// TIA Portal project "2022.06.14_通信方式" (V17)

(* hardware
DEVICE "S7-1200 station_1"  S7-1200 Station
   slot 0: "Rack_0"  S7-1200 Rack  Rack  V1.0
   slot 1: "PLC_1"  CPU 1212C DC/DC/DC  6ES7 212-1AE40-0XB0  V4.5
   slot 2: "AI 4x13BIT/AQ 2x14BIT_1"  SM 1234 AI4/AQ2  6ES7 234-4HE30-0XB0  V1.0
*)

// ===== PLC "PLC_1"  CPU 1212C DC/DC/DC =====

VAR_GLOBAL   // PLC tag table "默认变量表"
   "液位测量" AT %IW96 : Word;
   "百分比" AT %MD40 : DWord;
   "模拟量输出通道" AT %MD44 : UDInt;
   "所需频率(1)" AT %MD0 : Real;
   "压力2模拟输入通道" AT %IW100 : Int;
   "液位" AT %MD4 : Real;
   "频率" AT %MD8 : Real;
   "Tag_2" AT %MD12 : Real;
   "模拟量输出" AT %QW96 : Int;
   "设定液位值" AT %MD20 : Real;
   "实际液位值" AT %MD24 : Real;
   "轴_1_脉冲" AT %Q0.0 : Bool;
   "轴_1_方向" AT %Q0.1 : Bool;
   "轴_1_LowHwLimitSwitch" AT %I0.0 : Bool;
   "轴_1_HighHwLimitSwitch" AT %I0.1 : Bool;
   "轴_1_PassiveHomingSwitch" AT %I0.2 : Bool;
   "轴_1_归位开关" AT %I0.3 : Bool;
   "启用轴" AT %M0.0 : Bool;
   "完成位" AT %M0.1 : Bool;
   "Tag_1" AT %M0.2 : Bool;
   "回原点" AT %I1.0 : Bool;
   "Tag_3" AT %M0.4 : Bool;
   "Tag_4" AT %M0.5 : Bool;
   "Tag_5" AT %M0.3 : Bool;
   "触发绝对定位" AT %I1.1 : Bool;
   "Tag_7" AT %M0.6 : Bool;
   "指定位置" AT %MD30 : Real;
   "指定速度" AT %MD34 : Real;
   "Tag_6" AT %M0.7 : Bool;
   "Tag_8" AT %I1.2 : Bool;
   "Tag_9" AT %M1.0 : Bool;
   "触发相对位移指令" AT %I1.3 : Bool;
   "Tag_11" AT %M1.1 : Bool;
   "相对位置" AT %MD28 : Real;
   "速度" AT %MD32 : Real;
   "触发恒速" AT %I0.4 : Bool;
   "Tag_10" AT %M1.2 : Bool;
   "Tag_12" AT %MD36 : Real;
   "Tag_13" AT %I1.5 : Bool;
   "Tag_14" AT %M1.3 : Bool;
   "正点动" AT %I1.6 : Bool;
   "反点动" AT %I1.7 : Bool;
   "System_Byte" AT %MB100 : Byte;
   "FirstScan" AT %M100.0 : Bool;
   "DiagStatusUpdate" AT %M100.1 : Bool;
   "AlwaysTRUE" AT %M100.2 : Bool;
   "AlwaysFALSE" AT %M100.3 : Bool;
   "Tag_15" AT %M10.0 : Bool;
   "Tag_16" AT %M70.0 : Bool;
   "Tag_17" AT %M70.1 : Bool;
   "Tag_18" AT %M70.2 : Bool;
   "Clock_Byte" AT %MB10 : Byte;
   "Clock_10Hz" AT %M10.0 : Bool;
   "Clock_5Hz" AT %M10.1 : Bool;
   "Clock_2.5Hz" AT %M10.2 : Bool;
   "Clock_2Hz" AT %M10.3 : Bool;
   "Clock_1.25Hz" AT %M10.4 : Bool;
   "Clock_1Hz" AT %M10.5 : Bool;
   "Clock_0.625Hz" AT %M10.6 : Bool;
   "Clock_0.5Hz" AT %M10.7 : Bool;
END_VAR

DATA_BLOCK "发送数据"   // DB15
{ S7_Optimized_Access := 'FALSE' }
VERSION : 0.1
   VAR
      发送1 : Real;
      发送2 : Real;
      发送3 : Real;
      发送4 : Real;
   END_VAR
BEGIN
END_DATA_BLOCK

DATA_BLOCK "接收"   // DB18
{ S7_Optimized_Access := 'FALSE' }
VERSION : 0.1
   VAR
      接受1 : Real;
      接受2 : Real;
      接受3 : Real;
      接受4 : Real;
   END_VAR
BEGIN
END_DATA_BLOCK

// folder: System blocks/Program resources

DATA_BLOCK "IEC_Timer_0_DB"   // DB13
{ S7_Optimized_Access := 'TRUE' }
AUTHOR : Simatic
FAMILY : IEC
NAME : IEC_TMR
VERSION : 1.0
// stored: InstanceOfName IEC_TIMER
"IEC_TIMER"
BEGIN
END_DATA_BLOCK

// folder: (top level)

DATA_BLOCK "轴_1"   // DB2, Motion_DB
{ S7_Optimized_Access := 'TRUE' }
AUTHOR : SIMATIC
FAMILY : BasicMC
NAME : TO_PosAx
VERSION : 8.0
// stored: InstanceOfName TO_PositioningAxis
"TO_PositioningAxis"
BEGIN
   // Axis.HomingReferencePointSwitch_AddressCU = %I0.3
   // Axis.LengthUnitNormalized.Distance = 1013
   // Axis.PositionLimitsMax_AddressCU = %I0.1
   // Axis.PositionLimitsMin_AddressCU = %I0.0
   // Axis.OnlinePtoModeCU = 16#0000_0002
   // Axis.DirectionOutputEnabledCU = TRUE
   // Axis.SelectedChannel2EnumCU = %Q0.1
   // Axis.SelectedChannel1EnumCU = %Q0.0
   // Pulse.MinDeltaDeltaFrequencyCU = 0.004
   // Pulse.MaxDeltaDeltaFrequencyCU = 1.0E+10
   // Pulse.MinDeltaFrequencyCU = 0.005
   // Pulse.MaxDeltaFrequencyCU = 9.5E+9
   // Pulse.MinFrequencyCU = 1.0
   // Pulse.MaxFrequencyCU = 100000.0
   // Pulse.OutputSourceCU = 16#0000_0000
   // Axis.SelectPTO = 0
END_DATA_BLOCK

ORGANIZATION_BLOCK "Main"   // OB1, LAD, ProgramCycle
TITLE = "Main Program Sweep (Cycle)"
{ S7_Optimized_Access := 'TRUE' }
VERSION : 0.1
   VAR_INPUT
      Initial_Call : Bool;   // Initial call of this OB
      Remanence : Bool;   // =True, if remanent data are available
   END_VAR
BEGIN

REGION Network 1
   // 把1200的数据发送到smart的PLC中.DB1给smart。100是smart地址.属性中一定要取消优化块的访问
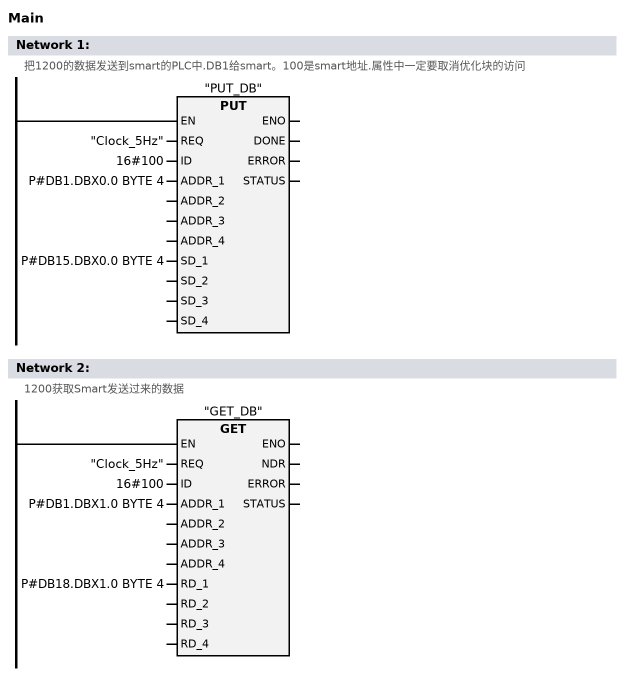
   "PUT_DB"(REQ := "Clock_5Hz", ID := 16#100, ADDR_1 := P#DB1.DBX0.0 BYTE 4, SD_1 := P#DB15.DBX0.0 BYTE 4);   // PUT
END_REGION

REGION Network 2
   // 1200获取Smart发送过来的数据
   "GET_DB"(REQ := "Clock_5Hz", ID := 16#100, ADDR_1 := P#DB1.DBX1.0 BYTE 4, RD_1 := P#DB18.DBX1.0 BYTE 4);   // GET
END_REGION
END_ORGANIZATION_BLOCK